(* PLC project Unnamed, Unknown Unnamed 1 *)
(* stored: creationDateTime 2025-05-14T12:21:41, modificationDateTime 2025-05-14T13:13:56 *)

(* in1 *)
PROGRAM traffic_light
  VAR
    in1 : BOOL;
    red : BOOL;
    yellow : BOOL;
    green : BOOL;
    timer : BOOL;
    TP0 : TP;
    TP2 : TP;
    TP3 : TP;
  END_VAR

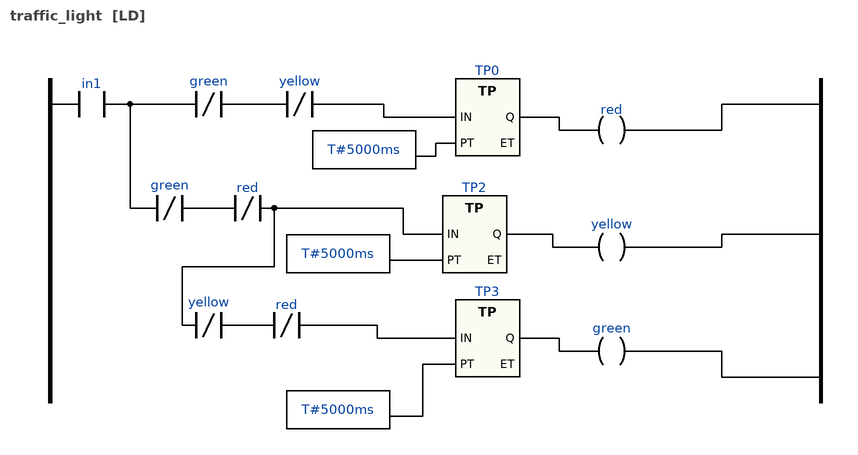
(* LD diagram, written out as Structured Text *)
TP0(IN := in1 AND NOT green AND NOT yellow, PT := T#5000ms);
red := TP0.Q;
TP2(IN := in1 AND NOT green AND NOT red, PT := T#5000ms);
yellow := TP2.Q;
TP3(IN := in1 AND NOT green AND NOT red AND NOT yellow AND NOT red, PT := T#5000ms);
green := TP3.Q;
END_PROGRAM

CONFIGURATION Config0
  RESOURCE Res0 ON PLC
    TASK task0(INTERVAL := T#20ms, PRIORITY := 0);
    PROGRAM instance0 WITH task0 : traffic_light;
  END_RESOURCE
END_CONFIGURATION
